(* Logix 5000 project; controller cal1632 1756-L62 rev 16.20; software revision 16.05; part 10 of 61 *)
(* tags used below, declared in another part *)
   FAULT : BOOL;
   p01_param_temp_limit : REAL;
   p01r09_pb_global_reset : BOOL;
   p02r11 : routine;
   p02r11_timer_fault : TIMER[4];
   p02r11_timer_warning : TIMER[4];
   p02r12 : routine;
   p02r12_timer_fault : TIMER[4];
   p02r12_timer_warning : TIMER[4];
   p02r13 : routine;
   p02r13_timer_fault : TIMER[4];
   p02r13_timer_warning : TIMER[4];
   p02r14 : routine;
   p02r14_timer_fault : TIMER[4];
   p02r14_timer_warning : TIMER[4];
   p02r15 : routine;
   p02r15_timer_fault : TIMER[4];
   p02r15_timer_warning : TIMER[4];
   p11_ai_prs : REAL;
   p11_ai_tc01 : REAL;
   p11_ai_tc02 : REAL;
   p11_dint_to_hmi : DINT[16];
   p11_param_shutdown_temp : REAL;
   p11_param_zone_pressure : REAL;
   p11r01 : routine;
   p11r02 : routine;
   p11r02_fault_exists : BOOL;
   p11r02_not_safe_temp : BOOL;
   p11r02_safe_temp : BOOL;
   p11r02_shutdown_temp : BOOL;
   p11r02_timer_fault : TIMER[4];
   p11r02_timer_safe_temp : TIMER[2];
   p11r02_timer_warning : TIMER[4];
   p11r02_unack_fault : BOOL;
   p11r02_unack_warning : BOOL;
   p11r02_warning_exists : BOOL;
   p11r03 : routine;
   p11r04 : routine;
   p11r05 : routine;
   p11r06 : routine;
   p11r07 : routine;
   p11r08 : routine;
   p11r09 : routine;
   p11r10 : routine;
   p11r20 : routine;
   p11r30 : routine;
   p11r30_pb_zone_off : BOOL;
   p11r31 : routine;
   p11r32 : routine;
(* P02_MOP_HMI_Iface, continued *)

ROUTINE R11   (* ladder *)
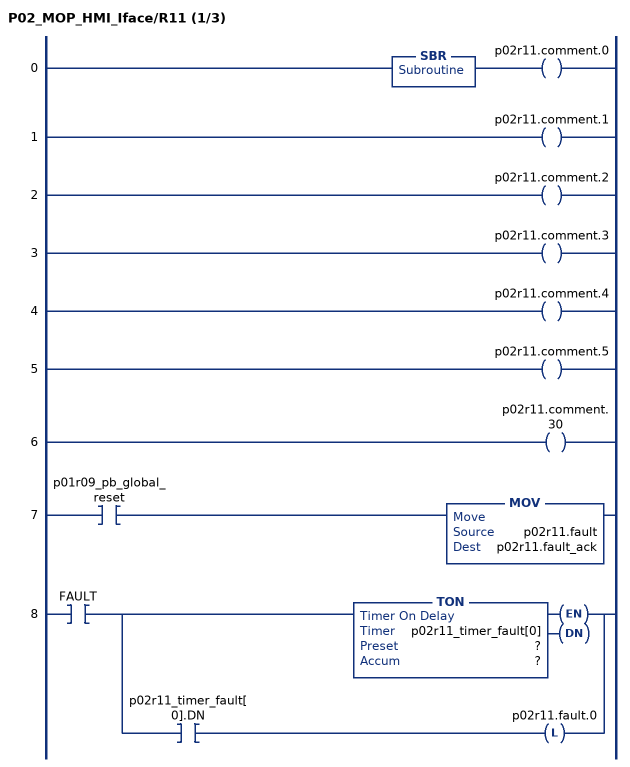
   0: SBR()OTE(p02r11.comment.0);
   1: OTE(p02r11.comment.1);
   2: OTE(p02r11.comment.2);
   3: OTE(p02r11.comment.3);
   4: OTE(p02r11.comment.4);
   5: OTE(p02r11.comment.5);
   6: OTE(p02r11.comment.30);
   7: XIC(p01r09_pb_global_reset)MOV(p02r11.fault,p02r11.fault_ack);
   8: XIC(FAULT)[TON(p02r11_timer_fault[0],?,?) ,XIC(p02r11_timer_fault[0].DN) OTL(p02r11.fault.0) ];
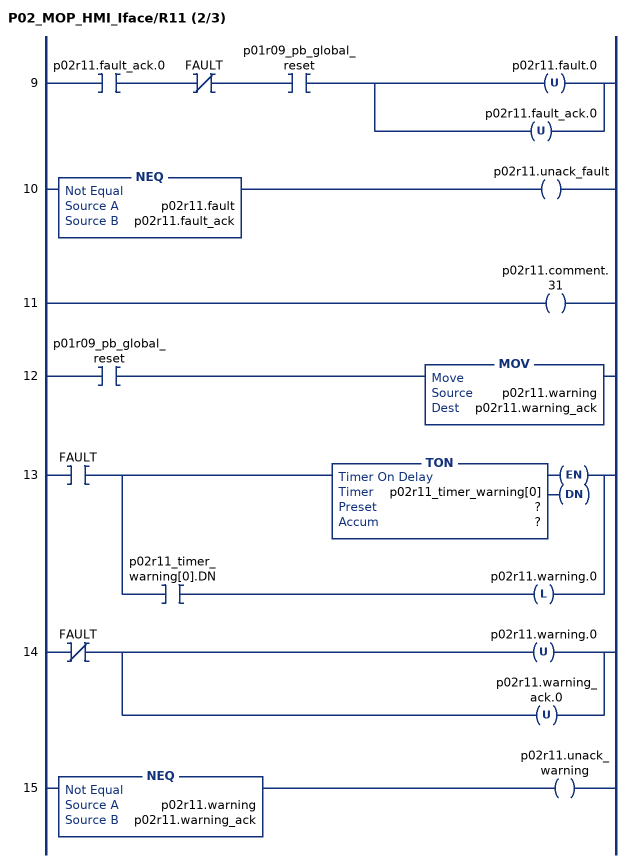
   9: XIC(p02r11.fault_ack.0)XIO(FAULT)XIC(p01r09_pb_global_reset)[OTU(p02r11.fault.0) ,OTU(p02r11.fault_ack.0) ];
   10: NEQ(p02r11.fault,p02r11.fault_ack)OTE(p02r11.unack_fault);
   11: OTE(p02r11.comment.31);
   12: XIC(p01r09_pb_global_reset)MOV(p02r11.warning,p02r11.warning_ack);
   13: XIC(FAULT)[TON(p02r11_timer_warning[0],?,?) ,XIC(p02r11_timer_warning[0].DN) OTL(p02r11.warning.0) ];
   14: XIO(FAULT)[OTU(p02r11.warning.0) ,OTU(p02r11.warning_ack.0) ];
   15: NEQ(p02r11.warning,p02r11.warning_ack)OTE(p02r11.unack_warning);
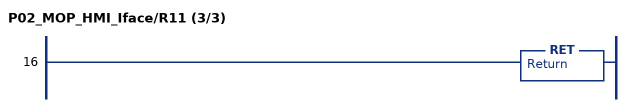
   16: RET();
END_ROUTINE

ROUTINE R12   (* ladder *)
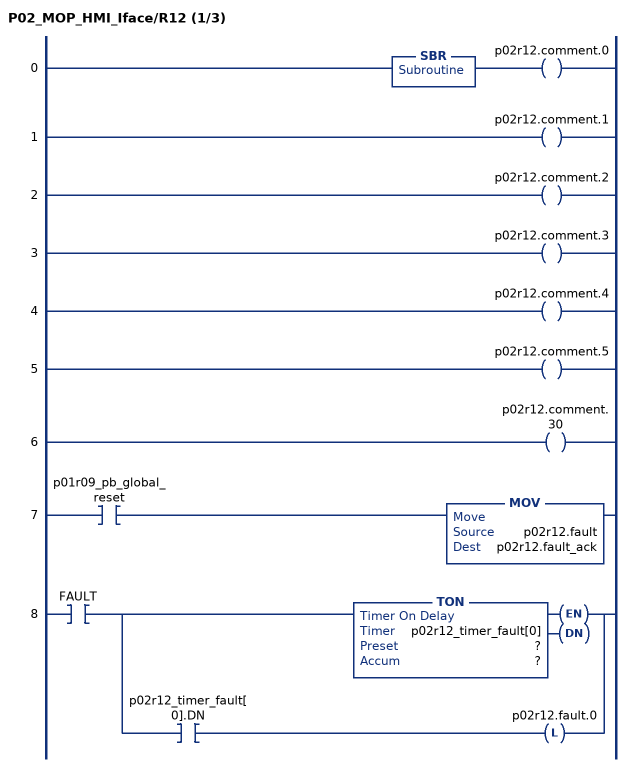
   0: SBR()OTE(p02r12.comment.0);
   1: OTE(p02r12.comment.1);
   2: OTE(p02r12.comment.2);
   3: OTE(p02r12.comment.3);
   4: OTE(p02r12.comment.4);
   5: OTE(p02r12.comment.5);
   6: OTE(p02r12.comment.30);
   7: XIC(p01r09_pb_global_reset)MOV(p02r12.fault,p02r12.fault_ack);
   8: XIC(FAULT)[TON(p02r12_timer_fault[0],?,?) ,XIC(p02r12_timer_fault[0].DN) OTL(p02r12.fault.0) ];
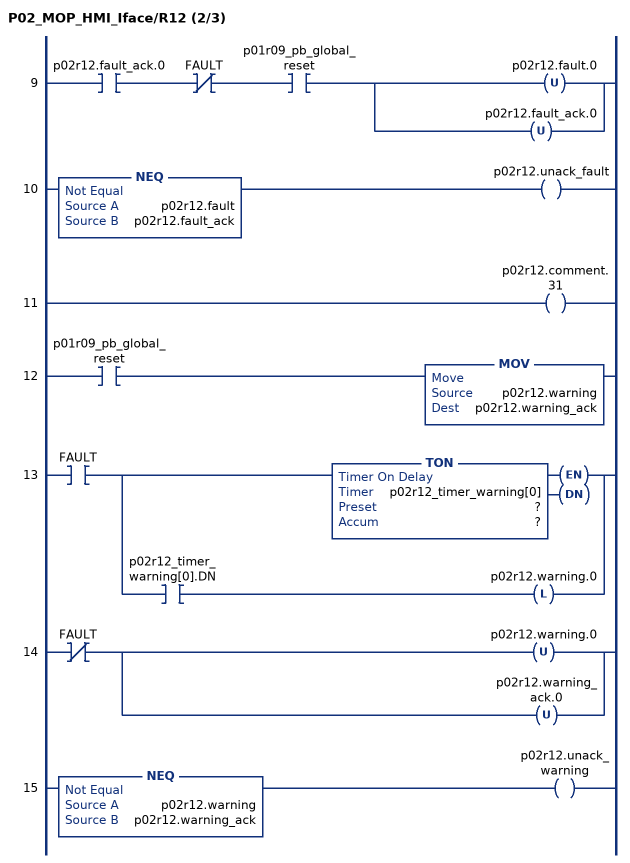
   9: XIC(p02r12.fault_ack.0)XIO(FAULT)XIC(p01r09_pb_global_reset)[OTU(p02r12.fault.0) ,OTU(p02r12.fault_ack.0) ];
   10: NEQ(p02r12.fault,p02r12.fault_ack)OTE(p02r12.unack_fault);
   11: OTE(p02r12.comment.31);
   12: XIC(p01r09_pb_global_reset)MOV(p02r12.warning,p02r12.warning_ack);
   13: XIC(FAULT)[TON(p02r12_timer_warning[0],?,?) ,XIC(p02r12_timer_warning[0].DN) OTL(p02r12.warning.0) ];
   14: XIO(FAULT)[OTU(p02r12.warning.0) ,OTU(p02r12.warning_ack.0) ];
   15: NEQ(p02r12.warning,p02r12.warning_ack)OTE(p02r12.unack_warning);
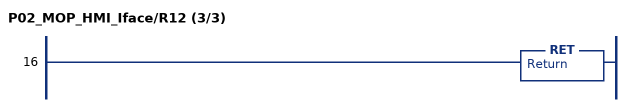
   16: RET();
END_ROUTINE

ROUTINE R13   (* ladder *)
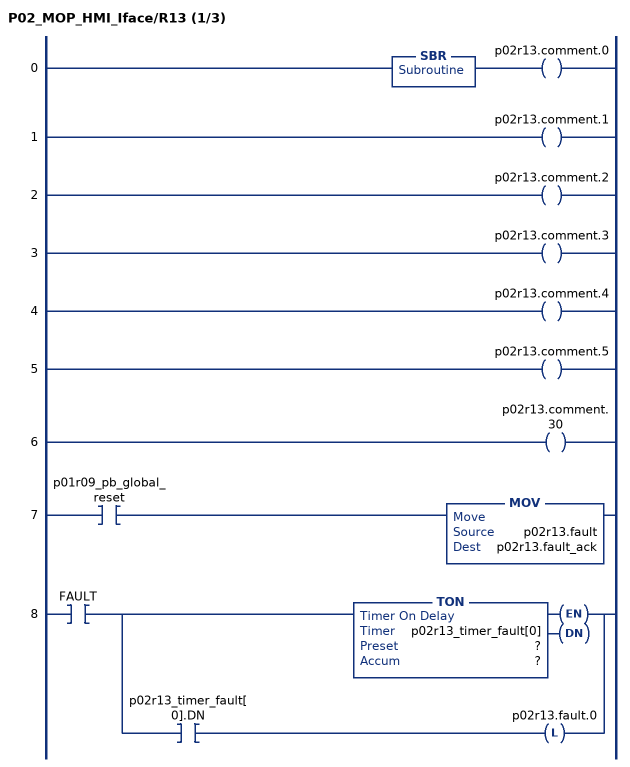
   0: SBR()OTE(p02r13.comment.0);
   1: OTE(p02r13.comment.1);
   2: OTE(p02r13.comment.2);
   3: OTE(p02r13.comment.3);
   4: OTE(p02r13.comment.4);
   5: OTE(p02r13.comment.5);
   6: OTE(p02r13.comment.30);
   7: XIC(p01r09_pb_global_reset)MOV(p02r13.fault,p02r13.fault_ack);
   8: XIC(FAULT)[TON(p02r13_timer_fault[0],?,?) ,XIC(p02r13_timer_fault[0].DN) OTL(p02r13.fault.0) ];
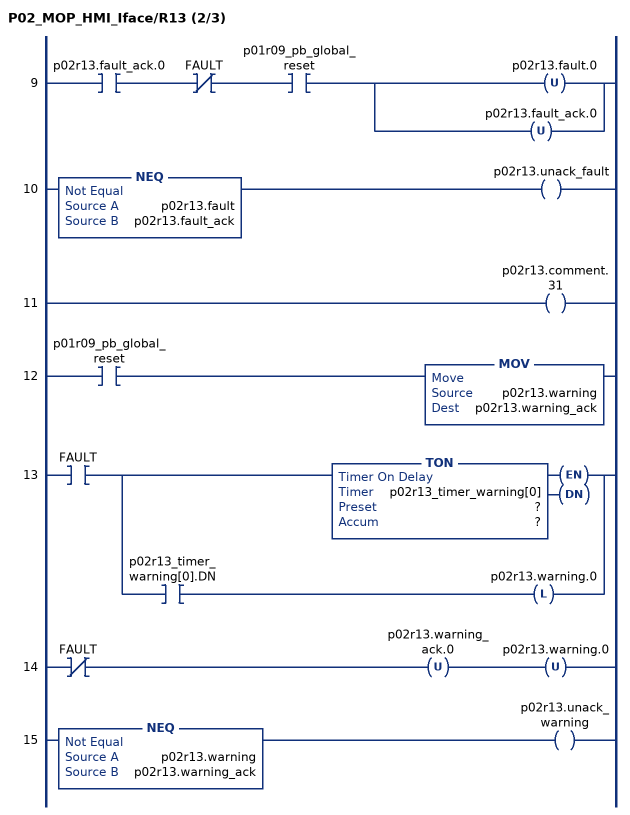
   9: XIC(p02r13.fault_ack.0)XIO(FAULT)XIC(p01r09_pb_global_reset)[OTU(p02r13.fault.0) ,OTU(p02r13.fault_ack.0) ];
   10: NEQ(p02r13.fault,p02r13.fault_ack)OTE(p02r13.unack_fault);
   11: OTE(p02r13.comment.31);
   12: XIC(p01r09_pb_global_reset)MOV(p02r13.warning,p02r13.warning_ack);
   13: XIC(FAULT)[TON(p02r13_timer_warning[0],?,?) ,XIC(p02r13_timer_warning[0].DN) OTL(p02r13.warning.0) ];
   14: XIO(FAULT)OTU(p02r13.warning_ack.0)OTU(p02r13.warning.0);
   15: NEQ(p02r13.warning,p02r13.warning_ack)OTE(p02r13.unack_warning);
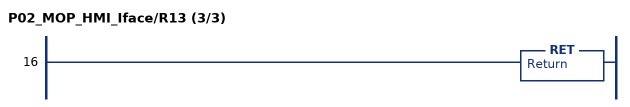
   16: RET();
END_ROUTINE

ROUTINE R14   (* ladder *)
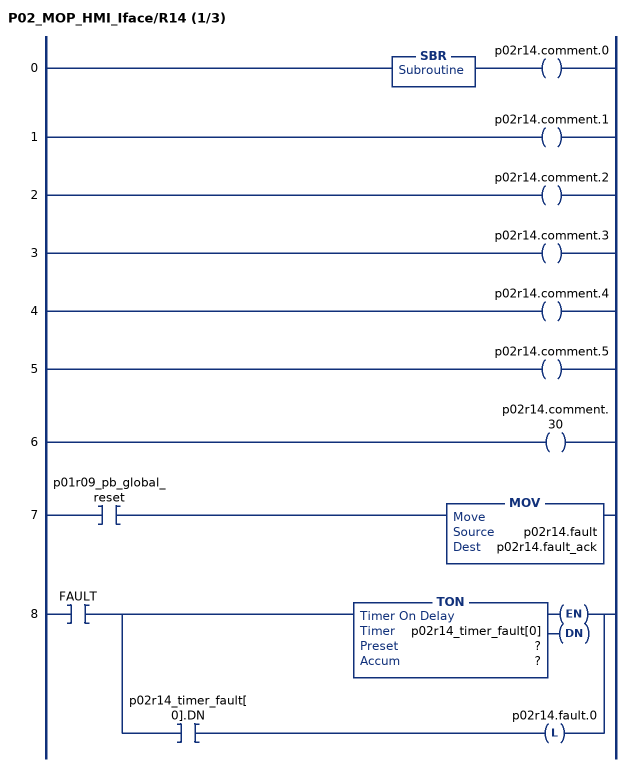
   0: SBR()OTE(p02r14.comment.0);
   1: OTE(p02r14.comment.1);
   2: OTE(p02r14.comment.2);
   3: OTE(p02r14.comment.3);
   4: OTE(p02r14.comment.4);
   5: OTE(p02r14.comment.5);
   6: OTE(p02r14.comment.30);
   7: XIC(p01r09_pb_global_reset)MOV(p02r14.fault,p02r14.fault_ack);
   8: XIC(FAULT)[TON(p02r14_timer_fault[0],?,?) ,XIC(p02r14_timer_fault[0].DN) OTL(p02r14.fault.0) ];
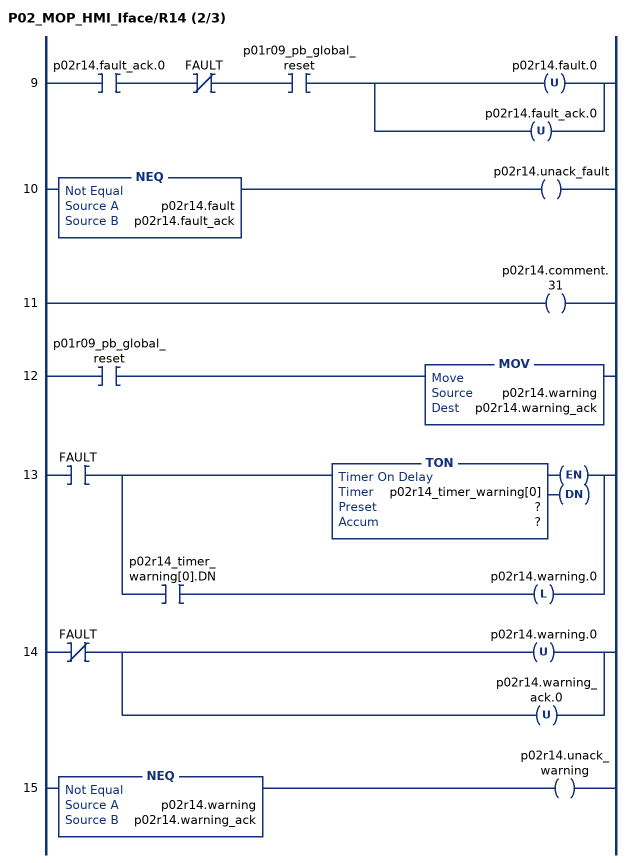
   9: XIC(p02r14.fault_ack.0)XIO(FAULT)XIC(p01r09_pb_global_reset)[OTU(p02r14.fault.0) ,OTU(p02r14.fault_ack.0) ];
   10: NEQ(p02r14.fault,p02r14.fault_ack)OTE(p02r14.unack_fault);
   11: OTE(p02r14.comment.31);
   12: XIC(p01r09_pb_global_reset)MOV(p02r14.warning,p02r14.warning_ack);
   13: XIC(FAULT)[TON(p02r14_timer_warning[0],?,?) ,XIC(p02r14_timer_warning[0].DN) OTL(p02r14.warning.0) ];
   14: XIO(FAULT)[OTU(p02r14.warning.0) ,OTU(p02r14.warning_ack.0) ];
   15: NEQ(p02r14.warning,p02r14.warning_ack)OTE(p02r14.unack_warning);
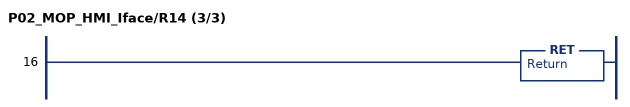
   16: RET();
END_ROUTINE

ROUTINE R15   (* ladder *)
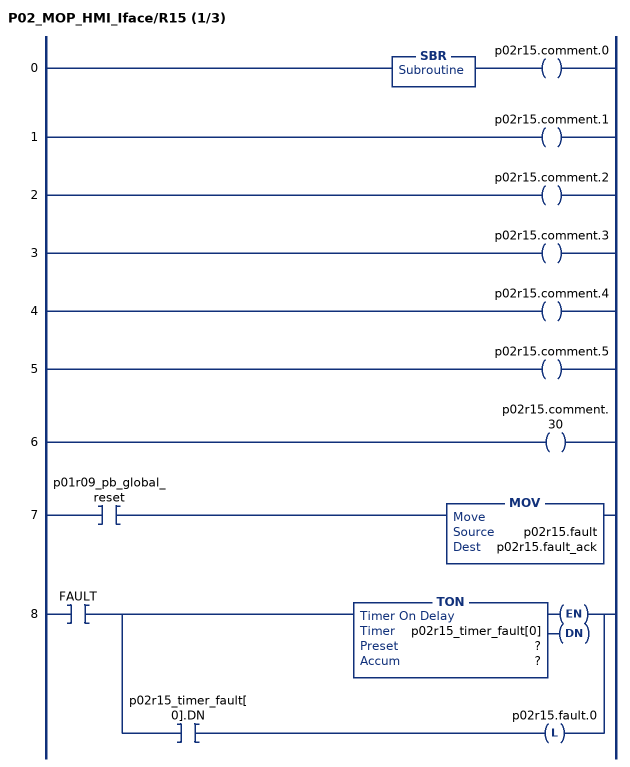
   0: SBR()OTE(p02r15.comment.0);
   1: OTE(p02r15.comment.1);
   2: OTE(p02r15.comment.2);
   3: OTE(p02r15.comment.3);
   4: OTE(p02r15.comment.4);
   5: OTE(p02r15.comment.5);
   6: OTE(p02r15.comment.30);
   7: XIC(p01r09_pb_global_reset)MOV(p02r15.fault,p02r15.fault_ack);
   8: XIC(FAULT)[TON(p02r15_timer_fault[0],?,?) ,XIC(p02r15_timer_fault[0].DN) OTL(p02r15.fault.0) ];
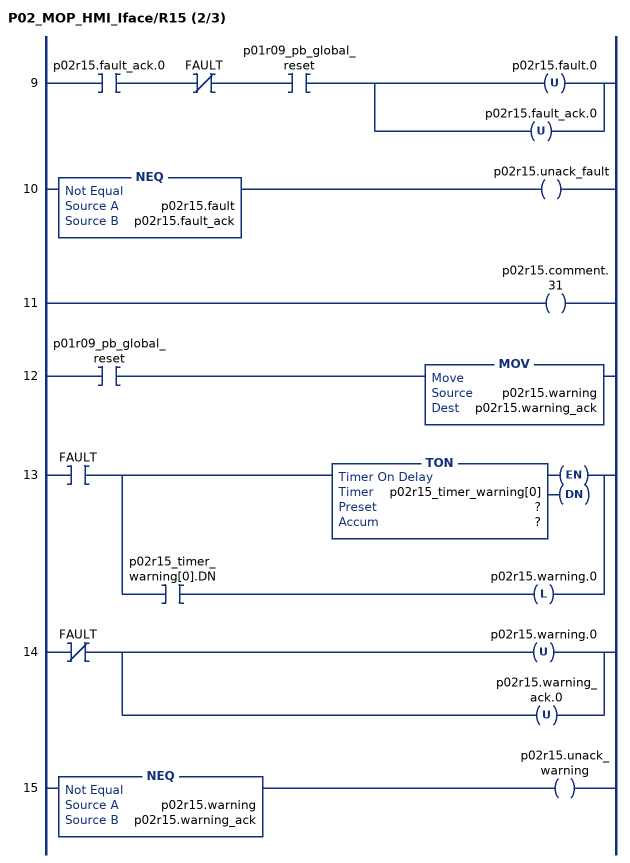
   9: XIC(p02r15.fault_ack.0)XIO(FAULT)XIC(p01r09_pb_global_reset)[OTU(p02r15.fault.0) ,OTU(p02r15.fault_ack.0) ];
   10: NEQ(p02r15.fault,p02r15.fault_ack)OTE(p02r15.unack_fault);
   11: OTE(p02r15.comment.31);
   12: XIC(p01r09_pb_global_reset)MOV(p02r15.warning,p02r15.warning_ack);
   13: XIC(FAULT)[TON(p02r15_timer_warning[0],?,?) ,XIC(p02r15_timer_warning[0].DN) OTL(p02r15.warning.0) ];
   14: XIO(FAULT)[OTU(p02r15.warning.0) ,OTU(p02r15.warning_ack.0) ];
   15: NEQ(p02r15.warning,p02r15.warning_ack)OTE(p02r15.unack_warning);
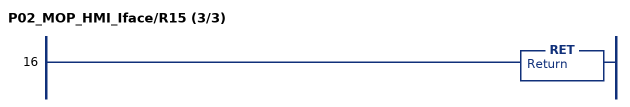
   16: RET();
END_ROUTINE
END_PROGRAM

PROGRAM P11_Zone_1   (* main routine R01_Main *)

ROUTINE R01_Main   (* ladder *)
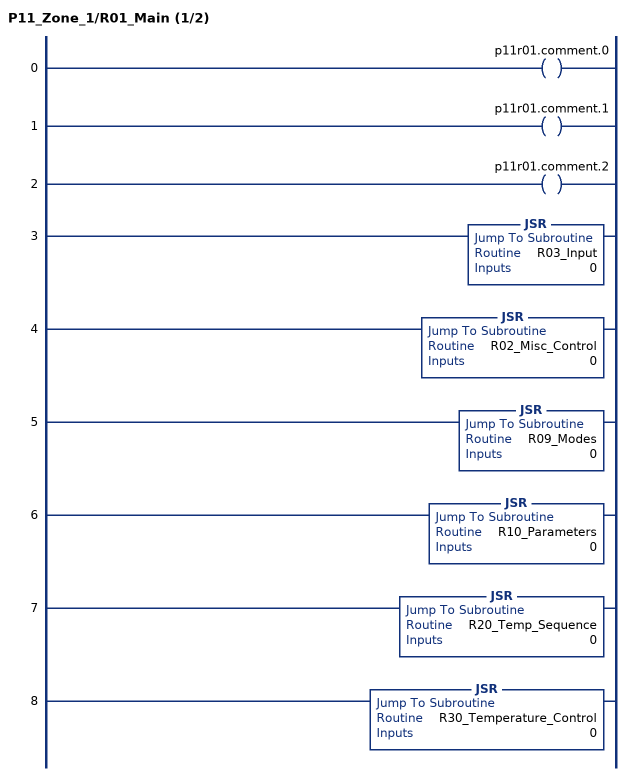
   0: OTE(p11r01.comment.0);
   1: OTE(p11r01.comment.1);
   2: OTE(p11r01.comment.2);
   3: JSR(R03_Input,0);
   4: JSR(R02_Misc_Control,0);
   5: JSR(R09_Modes,0);
   6: JSR(R10_Parameters,0);
   7: JSR(R20_Temp_Sequence,0);
   8: JSR(R30_Temperature_Control,0);
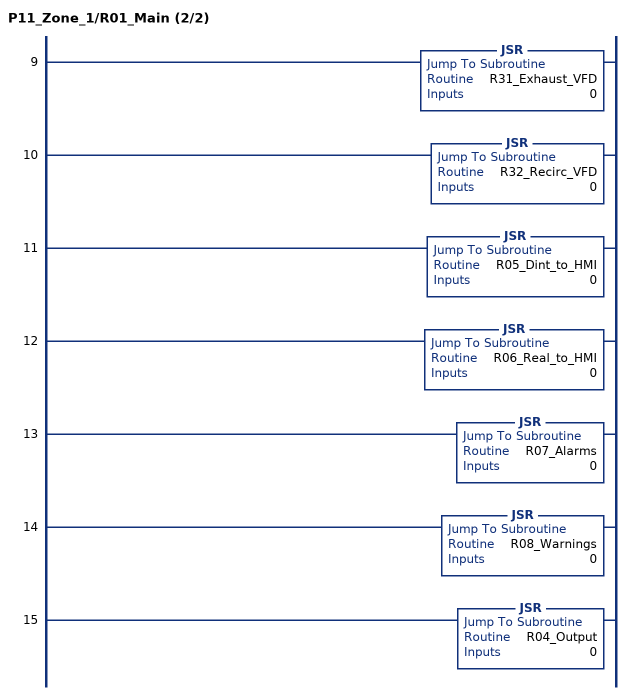
   9: JSR(R31_Exhaust_VFD,0);
   10: JSR(R32_Recirc_VFD,0);
   11: JSR(R05_Dint_to_HMI,0);
   12: JSR(R06_Real_to_HMI,0);
   13: JSR(R07_Alarms,0);
   14: JSR(R08_Warnings,0);
   15: JSR(R04_Output,0);
END_ROUTINE

ROUTINE R02_Misc_Control   (* ladder *)
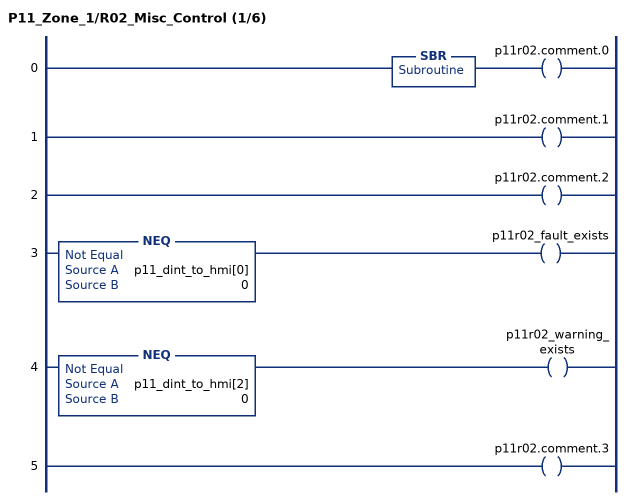
   0: SBR()OTE(p11r02.comment.0);
   1: OTE(p11r02.comment.1);
   2: OTE(p11r02.comment.2);
   3: NEQ(p11_dint_to_hmi[0],0)OTE(p11r02_fault_exists);
   4: NEQ(p11_dint_to_hmi[2],0)OTE(p11r02_warning_exists);
   5: OTE(p11r02.comment.3);
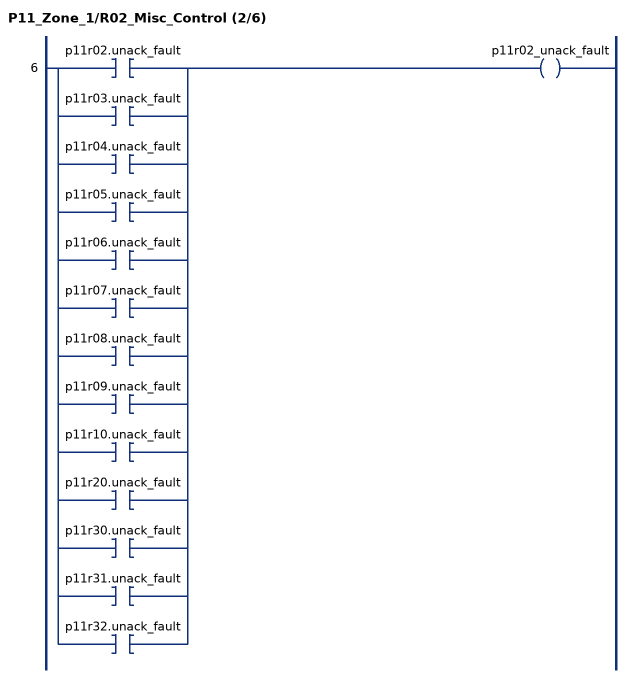
   6: [XIC(p11r02.unack_fault) ,XIC(p11r03.unack_fault) ,XIC(p11r04.unack_fault) ,XIC(p11r05.unack_fault) ,XIC(p11r06.unack_fault) ,XIC(p11r07.unack_fault) ,XIC(p11r08.unack_fault) ,XIC(p11r09.unack_fault) ,XIC(p11r10.unack_fault) ,XIC(p11r20.unack_fault) ,XIC(p11r30.unack_fault) ,XIC(p11r31.unack_fault) ,XIC(p11r32.unack_fault) ]OTE(p11r02_unack_fault);
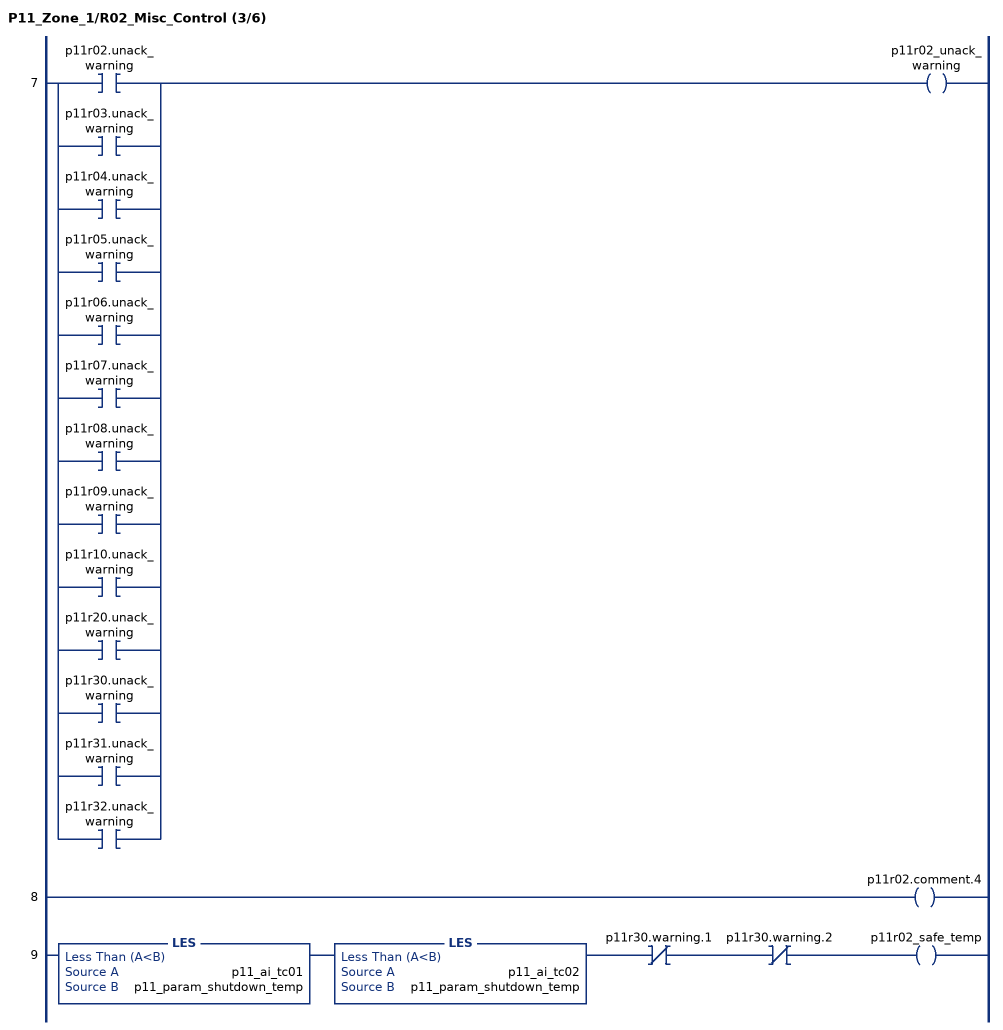
   7: [XIC(p11r02.unack_warning) ,XIC(p11r03.unack_warning) ,XIC(p11r04.unack_warning) ,XIC(p11r05.unack_warning) ,XIC(p11r06.unack_warning) ,XIC(p11r07.unack_warning) ,XIC(p11r08.unack_warning) ,XIC(p11r09.unack_warning) ,XIC(p11r10.unack_warning) ,XIC(p11r20.unack_warning) ,XIC(p11r30.unack_warning) ,XIC(p11r31.unack_warning) ,XIC(p11r32.unack_warning) ]OTE(p11r02_unack_warning);
   8: OTE(p11r02.comment.4);
   9: LES(p11_ai_tc01,p11_param_shutdown_temp)LES(p11_ai_tc02,p11_param_shutdown_temp)XIO(p11r30.warning.1)XIO(p11r30.warning.2)OTE(p11r02_safe_temp);
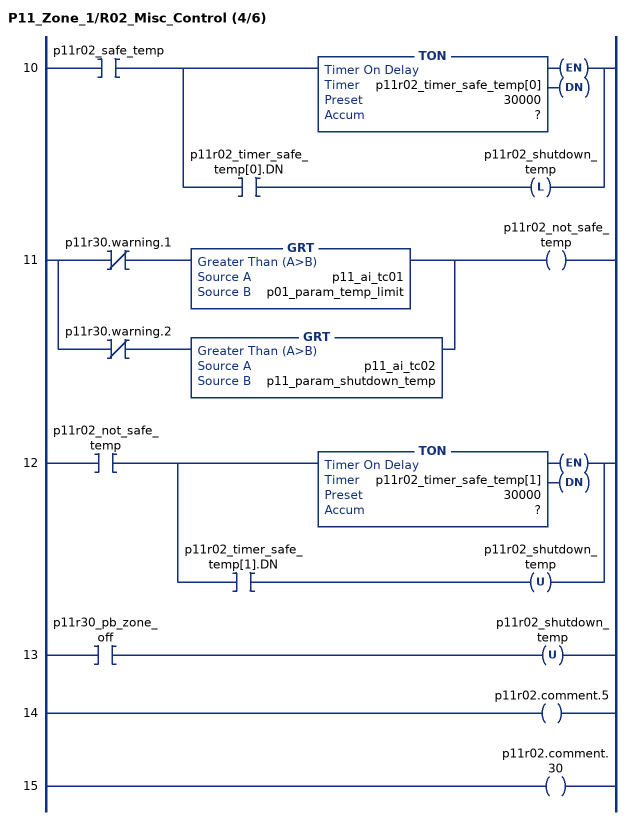
   10: XIC(p11r02_safe_temp)[TON(p11r02_timer_safe_temp[0],?,?) ,XIC(p11r02_timer_safe_temp[0].DN) OTL(p11r02_shutdown_temp) ];
   11: [XIO(p11r30.warning.1) GRT(p11_ai_tc01,p01_param_temp_limit) ,XIO(p11r30.warning.2) GRT(p11_ai_tc02,p11_param_shutdown_temp) ]OTE(p11r02_not_safe_temp);
   12: XIC(p11r02_not_safe_temp)[TON(p11r02_timer_safe_temp[1],?,?) ,XIC(p11r02_timer_safe_temp[1].DN) OTU(p11r02_shutdown_temp) ];
   13: XIC(p11r30_pb_zone_off)OTU(p11r02_shutdown_temp);
   14: OTE(p11r02.comment.5);
   15: OTE(p11r02.comment.30);
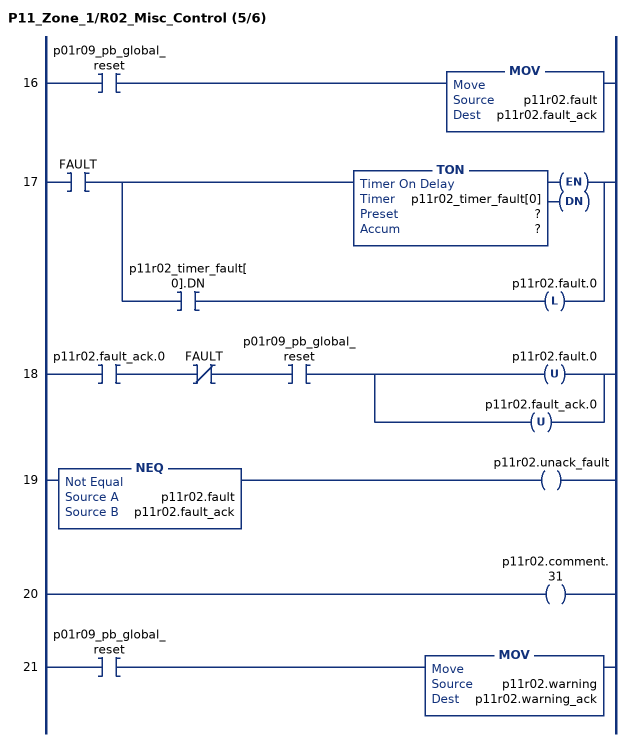
   16: XIC(p01r09_pb_global_reset)MOV(p11r02.fault,p11r02.fault_ack);
   17: XIC(FAULT)[TON(p11r02_timer_fault[0],?,?) ,XIC(p11r02_timer_fault[0].DN) OTL(p11r02.fault.0) ];
   18: XIC(p11r02.fault_ack.0)XIO(FAULT)XIC(p01r09_pb_global_reset)[OTU(p11r02.fault.0) ,OTU(p11r02.fault_ack.0) ];
   19: NEQ(p11r02.fault,p11r02.fault_ack)OTE(p11r02.unack_fault);
   20: OTE(p11r02.comment.31);
   21: XIC(p01r09_pb_global_reset)MOV(p11r02.warning,p11r02.warning_ack);
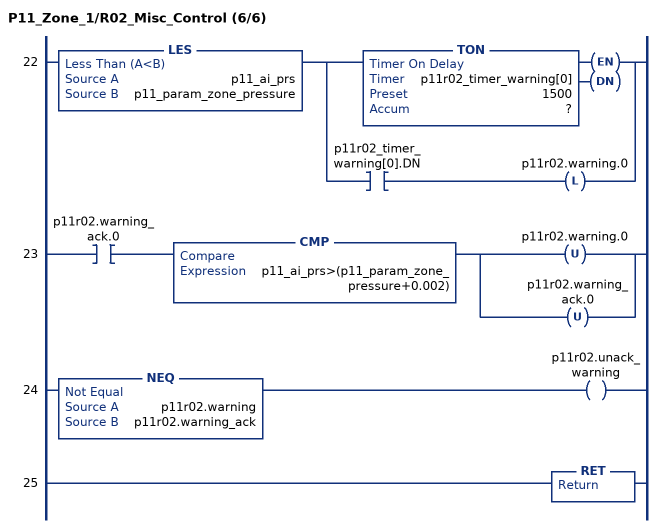
   22: LES(p11_ai_prs,p11_param_zone_pressure)[TON(p11r02_timer_warning[0],?,?) ,XIC(p11r02_timer_warning[0].DN) OTL(p11r02.warning.0) ];
   23: XIC(p11r02.warning_ack.0)CMP(p11_ai_prs>(p11_param_zone_pressure+0.002))[OTU(p11r02.warning.0) ,OTU(p11r02.warning_ack.0) ];
   24: NEQ(p11r02.warning,p11r02.warning_ack)OTE(p11r02.unack_warning);
   25: RET();
END_ROUTINE
